(* IEC 61131-3 sources: Persist/, 3 files *)

(* ---- Persist.typ ---- *)
(********************************************************************
 * COPYRIGHT --
 ********************************************************************
 * Library: Persist
 * File: Persist.typ
 * Author: davidblackburn
 * Created: October 04, 2013
 ********************************************************************
 * Data types of library Persist
 ********************************************************************)
(*Public types*)

TYPE
	PERSIST_ERR_enum :
		(
		PERSIST_ERR_INVALIDINPUT := 50000,
		PERSIST_ERR_OUTOFMEMORY,
		PERSIST_ERR_DATAMOVED_CHANGED
		);
	Persistence_Var_Metadata : 	STRUCT
		workingVariable : STRING[80];
		variableSize : UDINT;
		lastFileBackupTime : DATE_AND_TIME;
		dataChanged : BOOL;
		pSelf : UDINT;
	END_STRUCT;
	Persistence_Int_VarInfo_typ : 	STRUCT
		pMetadata : REFERENCE TO Persistence_Var_Metadata;
		pWorkingVariable : UDINT;
		sizeofWorkingVariable : UDINT;
		pPersistentMemory : UDINT;
	END_STRUCT;
	Persistence_Internal_typ : 	STRUCT
		WorkingVariableInfo : ARRAY[0..PERSIST_MAI_VARLIST]OF Persistence_Int_VarInfo_typ;
		ValidWorkingVariable : Persistence_Int_VarInfo_typ;
		iVariable : USINT;
		DataValid : BOOL;
	END_STRUCT;
	Persistence_OUT_STAT_typ : 	STRUCT
		RequiredMemory : UDINT; (*Number of bytes required to store every variable in WorkingVariableList*)
		Initialized : BOOL;
		Error : BOOL;
		ErrorID : UINT;
		ErrorString : STRING[PERSIST_STRLEN_ERRORSTRING];
	END_STRUCT;
	Persistence_OUT_typ : 	STRUCT
		STAT : Persistence_OUT_STAT_typ;
	END_STRUCT;
	Persistence_IN_typ : 	STRUCT
		pPersistentVariable : UDINT; (*Address of the persistent variable*)
		sizeofPersistentVariable : UDINT; (*Size of the persistent variable*)
		pDataValid : UDINT; (*Address of the DataValid variable. If *pDataValid == TRUE, then persistent memory is copied to working memory on startup. If *pDataValid == FALSE, then persistent memory is NOT copied to working memory*)
		WorkingVariableList : ARRAY[0..PERSIST_MAI_VARLIST]OF STRING[PERSIST_STRLEN_VARNAME]; (*List of working variables to be managed*)
	END_STRUCT;
	Persistence_typ : 	STRUCT
		IN : Persistence_IN_typ;
		OUT : Persistence_OUT_typ;
		Internal : Persistence_Internal_typ;
	END_STRUCT;
END_TYPE

(* ---- Persist.fun ---- *)
(********************************************************************
 * COPYRIGHT --
 ********************************************************************
 * Library: Persist
 * File: Persist.fun
 * Author: davidblackburn
 * Created: October 04, 2013
 ********************************************************************
 * Functions and function blocks of library Persist
 ********************************************************************)

FUNCTION PersistFn_Init : UINT (*Copy values from persistent memory to working memory*) (*$GROUP=User*)
	VAR_IN_OUT
		Persistence : Persistence_typ;
	END_VAR
END_FUNCTION

FUNCTION PersistFn_Cyclic : UINT (*Copy values from working memory to persistent memory*) (*$GROUP=User*)
	VAR_IN_OUT
		Persistence : Persistence_typ;
	END_VAR
END_FUNCTION

FUNCTION persistInternalMapMemory : UINT (*Internal: Determine memory addresses*) (*$GROUP=User*)
	VAR_IN_OUT
		Persistence : Persistence_typ;
	END_VAR
END_FUNCTION

FUNCTION persistInternalBackup : UINT (*Internal: Backup to persistent memory*) (*$GROUP=User*)
	VAR_IN_OUT
		Persistence : Persistence_typ;
	END_VAR
END_FUNCTION

FUNCTION persistInternalRestore : UINT (*Internal: Restore from persistent memory*) (*$GROUP=User*)
	VAR_IN_OUT
		Persistence : Persistence_typ;
	END_VAR
END_FUNCTION

FUNCTION persistUpdateMetadata : UINT
	VAR_INPUT
		Persistence : Persistence_typ;
	END_VAR
END_FUNCTION

(* ---- Persist.var ---- *)
(********************************************************************
 * COPYRIGHT --
 ********************************************************************
 * Library: Persist
 * File: Persist.var
 * Author: davidblackburn
 * Created: October 04, 2013
 ********************************************************************
 * Constants of library Persist
 ********************************************************************)
VAR CONSTANT
	PERSIST_MAI_VARLIST : USINT := 99;
	PERSIST_STRLEN_VARNAME : USINT := 120;
	PERSIST_STRLEN_ERRORSTRING : UINT := 320;
END_VAR
